{attribute 'linkalways'} 
{attribute 'no_explicit_call' := 'This FB is a CLASS and must be accessed using methods or properties'}
{attribute 'enable_dynamic_creation'}
FUNCTION_BLOCK Node_F_VN_MinElementElementwise_TcVnVector4_INT EXTENDS VisionNode
VAR
    ipContainer : _ITcVnContainer;
    aMin : _TcVnVector4_INT;
    hrPrev : _HRESULT(S_OK);
    hresult : _HRESULT(S_OK);
END_VAR

METHOD PUBLIC  Clone : I_Node
VAR
	pNode : POINTER TO Node_F_VN_MinElementElementwise_TcVnVector4_INT;
END_VAR
pNode := __NEW(Node_F_VN_MinElementElementwise_TcVnVector4_INT);
Clone := pNode^;
END_METHOD

METHOD FB_init : BOOL
VAR_INPUT
	bInitRetains : BOOL; // if TRUE, the retain variables are initialized (warm start / cold start)
	bInCopyCode : BOOL;  // if TRUE, the instance afterwards gets moved into the copy code (online change)
END_VAR
AddInput('ipContainer', ipContainer);
AddInput('aMin', aMin);
AddInput('hrPrev', hrPrev);
AddOutput('ipContainer', ipContainer);
AddOutput('hresult',hresult);
END_METHOD

METHOD PROTECTED OnExecute : HRESULT
hresult.Value := F_VN_MinElementElementwise_TcVnVector4_INT(
    ipContainer := ipContainer.Value,
    aMin := aMin.Value,
    hrPrev:= hrPrev.Value);
END_METHOD

METHOD PUBLIC PreExecutionCheck
VAR_INPUT
	Check : I_PreExecutionChecks;
END_VAR
Check.IsTrue(ipContainer.IsValid, 'ipContainer must be a valid container');
END_METHOD

END_FUNCTION_BLOCK

(* stored: Version 1.1.0.1, ProductVersion 3.1.4024.13
   POU Node_F_VN_MinElementElementwise_TcVnVector4_INT: Id {abca74b2-1f38-43ca-aa87-00498224dddf}, SpecialFunc None
   Folder Constructor: Id {9b80084a-e2ed-426c-83ee-c9fedbbadd57}
   Method Clone: Id {63bffaac-8363-4421-aae7-bea055286de2}
   Method FB_init: Id {2490808e-1413-4b43-9c4e-a8a9de6ca0e4}
   Method OnExecute: Id {b70943e4-9248-48c4-8dac-d37574a66c06}
   Method PreExecutionCheck: Id {cb51a488-a533-49ae-8be0-770c08cbe3e9} *)
